TYPE IO :
STRUCT
MesEventCode : ARRAY[1..7] OF WORD ; (*Akuo AlarmCode*)

END_STRUCT
END_TYPE

(* stored: Version 1.1.0.1, ProductVersion 3.1.4024.6
   DUT IO: Id {b01a5d24-6730-4dfe-a526-8523a4e88940} *)
